// TIA Portal V20 export
TYPE "typeCmControlNodeSoftCam"
// stored: Namespace Unit1.Em4
   STRUCT
      positionMoving { ExternalWritable := 'False'} : "Unit1.Em4.typeCmControlNodeSoftCamPositionMoving";
   END_STRUCT;
END_TYPE
